FUNCTION_BLOCK START
  (* Standard: 61499-2 *)
  (* Version 11-01-12, GASR *)
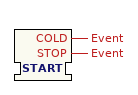
  EVENT_OUTPUT
    COLD;
    STOP;
  END_EVENT
  EC_STATES
    START;
  END_STATES
END_FUNCTION_BLOCK
